FUNCTION_BLOCK FB_GCSpinAxisJogServices EXTENDS FB_PackMLBase IMPLEMENTS I_ModuleServiceProperty
VAR_INPUT
	Ctrl : REFERENCE TO ST_GCSpinAxisJogCtrl;
	Status : REFERENCE TO ST_GCSpinAxisJogStatus;
	Axis_BaseUnit : REFERENCE TO FB_AxisControl;
END_VAR

VAR_OUTPUT
END_VAR

VAR
	_StartOneShot	: R_TRIG;
	_ResetOneShot	: R_TRIG;
	_StopOneShot	: R_TRIG;
	_AbortOneShot	: R_TRIG;
	
	_ModuleMode		: T_PackMLMode;
END_VAR

// Update service state
Status.State := stOut.eStateCurrent;

A00_TrigCommand();

SUPER^();

ACTION A00_TrigCommand:
_StartOneShot(CLK:= Ctrl.Start);
IF _StartOneShot.Q THEN
	RequestCommand(E_PackMLCommand.Start);
END_IF

_ResetOneShot(CLK:= Ctrl.Reset);
IF _ResetOneShot.Q THEN
	RequestCommand(E_PackMLCommand.Reset);
END_IF

_StopOneShot(CLK:= Ctrl.Stop);
IF _StopOneShot.Q THEN
	RequestCommand(E_PackMLCommand.Stop);
END_IF

_AbortOneShot(CLK:= Ctrl.Abort);
IF _AbortOneShot.Q THEN
	RequestCommand(E_PackMLCommand.Abort);
END_IF
END_ACTION

METHOD PROTECTED H_OnAborted
VAR_INPUT
	bFirstScan	: BOOL;
END_VAR
// Default action hook intentionally empty. Override in derived FBs when needed.
Status.Busy := FALSE;
Status.Done := FALSE;
Status.Aborted := TRUE;

RequestCommand(E_PackMLCommand.Clear);
END_METHOD

METHOD PROTECTED H_OnAborting : E_PackMLHookResult
VAR_INPUT
	bFirstScan	: BOOL;
END_VAR
Axis_BaseUnit.M_Jog(
	JogForward:= FALSE, 
	JogBackwards:= FALSE, 
	Mode:= Ctrl.Param.Mode,
	Position:= Ctrl.Param.Position,
	Velocity:= Ctrl.Param.Velocity,
	Acceleration:= Ctrl.Param.Acceleration,
	Deceleration:= Ctrl.Param.Deceleration);

H_OnAborting := E_PackMLHookResult.Done;
END_METHOD

METHOD PROTECTED H_OnClearing : E_PackMLHookResult
VAR_INPUT
	bFirstScan	: BOOL;
END_VAR

VAR
	bServoOn : BOOL;
	bError : BOOL;
	nErrorId : UDINT;
END_VAR
H_OnClearing := E_PackMLHookResult.Done;
END_METHOD

METHOD PROTECTED H_OnComplete
VAR_INPUT
	bFirstScan	: BOOL;
END_VAR
Status.Busy := FALSE;
Status.Done := TRUE;
Status.Error := FALSE;
Status.Aborted := FALSE;
Status.ErrorId := E_GCSpinAxisJogErrorCode.None;

IF NOT Ctrl.Start THEN
	RequestCommand(E_PackMLCommand.Reset);
END_IF
END_METHOD

METHOD PROTECTED H_OnCompleting : E_PackMLHookResult
VAR_INPUT
	bFirstScan	: BOOL;
END_VAR
Status.Busy := FALSE;
Status.Done := TRUE;
Status.Error := FALSE;
Status.Aborted := FALSE;
Status.ErrorId := E_GCSpinAxisJogErrorCode.None;

Axis_BaseUnit.M_Jog(
	JogForward:= FALSE, 
	JogBackwards:= FALSE, 
	Mode:= Ctrl.Param.Mode,
	Position:= Ctrl.Param.Position,
	Velocity:= Ctrl.Param.Velocity,
	Acceleration:= Ctrl.Param.Acceleration,
	Deceleration:= Ctrl.Param.Deceleration);

H_OnCompleting := E_PackMLHookResult.Done;
END_METHOD

METHOD PROTECTED H_OnExecute : E_PackMLHookResult
VAR_INPUT
	bFirstScan	: BOOL;
END_VAR

VAR
	bDone : BOOL;
	bError : BOOL;
END_VAR
H_OnExecute := E_PackMLHookResult.Busy;

Status.Busy := TRUE;
Status.Done := FALSE;
Status.Error := FALSE;
Status.Aborted := FALSE;
Status.ErrorId := E_GCSpinAxisJogErrorCode.None;

Axis_BaseUnit.M_Jog(
	JogForward:= Ctrl.Param.JogForward,
	JogBackwards:= Ctrl.Param.JogBackwards,
	Mode:= Ctrl.Param.Mode,
	Position:= Ctrl.Param.Position,
	Velocity:= Ctrl.Param.Velocity,
	Acceleration:= Ctrl.Param.Acceleration,
	Deceleration:= Ctrl.Param.Deceleration,
	Done=> bDone, Error=> bError);


IF Ctrl.Param.Mode = E_JogMode.MC_JOGMODE_INCHING THEN
	IF bDone THEN
		Status.Busy := FALSE;
		Status.Done := TRUE;
		H_OnExecute := E_PackMLHookResult.Done;
		RETURN;
	END_IF
END_IF

IF bError THEN
		Status.Error := TRUE;
		Status.ErrorId := E_GCSpinAxisJogErrorCode.Jog_Error_During_Execute;
		
		RequestCommand(E_PackMLCommand.Stop);
END_IF
END_METHOD

METHOD PROTECTED H_OnHeld
VAR_INPUT
	bFirstScan	: BOOL;
END_VAR
// Default action hook intentionally empty. Override in derived FBs when needed.
END_METHOD

METHOD PROTECTED H_OnHolding : E_PackMLHookResult
VAR_INPUT
	bFirstScan	: BOOL;
END_VAR
// Default transient hooks complete immediately; override when work is required.
H_OnHolding := E_PackMLHookResult.Done;
END_METHOD

METHOD PROTECTED H_OnIdle
VAR_INPUT
	bFirstScan	: BOOL;
END_VAR
// Default action hook intentionally empty. Override in derived FBs when needed.
Status.Busy := FALSE;
Status.Done := FALSE;
Status.Error := FALSE;
Status.Aborted := FALSE;
Status.ErrorId := E_GCSpinAxisJogErrorCode.None;
END_METHOD

METHOD PROTECTED H_OnResetting : E_PackMLHookResult
VAR_INPUT
	bFirstScan	: BOOL;
END_VAR
Status.Busy := FALSE;
Status.Done := FALSE;
Status.Error := FALSE;
Status.Aborted := FALSE;
Status.ErrorId := E_GCSpinAxisJogErrorCode.None;

H_OnResetting := E_PackMLHookResult.Done;
END_METHOD

METHOD PROTECTED H_OnStarting : E_PackMLHookResult
VAR_INPUT
	bFirstScan	: BOOL;
END_VAR
H_OnStarting := E_PackMLHookResult.Busy;

Status.Busy := TRUE;
Status.Done := FALSE;
Status.Error := FALSE;
Status.Aborted := FALSE;
Status.ErrorId := E_GCSpinAxisJogErrorCode.None;

// Check is servo on
IF Axis_BaseUnit.AxisStatus.Disabled THEN
	
	// Throw up error
	Status.Error:= TRUE;
	Status.ErrorId:= E_GCSpinAxisJogErrorCode.Axis_Not_Servo_On_During_Starting;
	
	// Request abort command
	RequestCommand(E_PackMLCommand.Abort);
	RETURN;
END_IF

// Check is axis not busy
IF Axis_BaseUnit.AxisStatus.HasJob THEN
	// Throw up error
	Status.Error:= TRUE;
	Status.ErrorId:= E_GCSpinAxisJogErrorCode.Axis_Is_Busy_During_Starting;
	
	// Request abort command
	RequestCommand(E_PackMLCommand.Stop);
	RETURN;
END_IF

// Check is param valid
IF (Ctrl.Param.JogBackwards AND Ctrl.Param.JogForward) OR
	(NOT Ctrl.Param.JogBackwards AND NOT Ctrl.Param.JogForward) OR
	Ctrl.Param.Velocity = 0 THEN
	// Throw up error
	Status.Error:= TRUE;
	Status.ErrorId:= E_GCSpinAxisJogErrorCode.Invalid_Param;
	
	// Request abort command
	RequestCommand(E_PackMLCommand.Stop);
	RETURN;
END_IF

H_OnStarting := E_PackMLHookResult.Done;
END_METHOD

METHOD PROTECTED H_OnStopped
VAR_INPUT
	bFirstScan	: BOOL;
END_VAR
// Default action hook intentionally empty. Override in derived FBs when needed.
Status.Busy := FALSE;
Status.Done := FALSE;
Status.Aborted := TRUE;
END_METHOD

METHOD PROTECTED H_OnStopping : E_PackMLHookResult
VAR_INPUT
	bFirstScan	: BOOL;
END_VAR
Axis_BaseUnit.M_Jog(
	JogForward:= FALSE, 
	JogBackwards:= FALSE, 
	Mode:= Ctrl.Param.Mode,
	Position:= Ctrl.Param.Position,
	Velocity:= Ctrl.Param.Velocity,
	Acceleration:= Ctrl.Param.Acceleration,
	Deceleration:= Ctrl.Param.Deceleration);

H_OnStopping := E_PackMLHookResult.Done;
END_METHOD

METHOD PROTECTED H_OnSuspended
VAR_INPUT
	bFirstScan	: BOOL;
END_VAR
// Default action hook intentionally empty. Override in derived FBs when needed.
END_METHOD

METHOD PROTECTED H_OnSuspending : E_PackMLHookResult
VAR_INPUT
	bFirstScan	: BOOL;
END_VAR
// Default transient hooks complete immediately; override when work is required.
H_OnSuspending := E_PackMLHookResult.Done;
END_METHOD

METHOD PROTECTED H_OnUndefined : E_PackMLHookResult
VAR_INPUT
	bFirstScan	: BOOL;
END_VAR
// The base FB leaves Undefined immediately unless a derived FB delays startup.
H_OnUndefined := E_PackMLHookResult.Done;
END_METHOD

METHOD PROTECTED H_OnUnholding : E_PackMLHookResult
VAR_INPUT
	bFirstScan	: BOOL;
END_VAR
// Default transient hooks complete immediately; override when work is required.
H_OnUnholding := E_PackMLHookResult.Done;
END_METHOD

METHOD PROTECTED H_OnUnsuspending : E_PackMLHookResult
VAR_INPUT
	bFirstScan	: BOOL;
END_VAR
// Default transient hooks complete immediately; override when work is required.
H_OnUnsuspending := E_PackMLHookResult.Done;
END_METHOD

PROPERTY ModuleMode : T_PackMLMode
GET
ModuleMode := _ModuleMode;
END_GET
SET
_ModuleMode := ModuleMode;
END_SET
END_PROPERTY

END_FUNCTION_BLOCK

(* stored: Version 1.1.0.1, ProductVersion 3.1.4026.18
   POU FB_GCSpinAxisJogServices: Id {a61ac5cd-09b6-4f2d-bc54-d014db7401a2}, SpecialFunc None
   Folder StateAction: Id {30486db3-fa54-4a70-b426-5f8ba9d0504f}
   Action A00_TrigCommand: Id {d9012b4d-3f7d-455a-a3d6-1f5152c45f28}
   Method H_OnAborted: Id {b48428e2-059a-4878-a27b-576d41f2ba26}
   Method H_OnAborting: Id {df4c7f2d-8a88-4d35-a321-0716e918b536}
   Method H_OnClearing: Id {9a60118e-19f9-4bca-893b-e890bf0b19c9}
   Method H_OnComplete: Id {fd680a59-d09e-4091-ac1f-b02ebd6a48e6}
   Method H_OnCompleting: Id {61491643-adf6-4106-831a-f4dfe9e14738}
   Method H_OnExecute: Id {2dba6e2e-7918-46c6-a0b6-50da9e5cf338}
   Method H_OnHeld: Id {fc1df435-3bb5-4a7c-8ab6-c741096bcbf0}
   Method H_OnHolding: Id {ece160eb-a5c7-4980-a6c1-7b10ad25762b}
   Method H_OnIdle: Id {801e1204-bf1d-4d12-b7fd-e2791384226a}
   Method H_OnResetting: Id {cd0cb289-d0f8-442c-af15-52d2005bf619}
   Method H_OnStarting: Id {bcd7c333-82d2-481d-9c52-d49b2030a18e}
   Method H_OnStopped: Id {7643e72d-21d0-42a9-a466-1828d294ec10}
   Method H_OnStopping: Id {7e40e9e4-ecf0-49b7-86b3-13897394333e}
   Method H_OnSuspended: Id {e85e43db-649a-4658-a8a4-46ee44393ec1}
   Method H_OnSuspending: Id {e203e9d4-d997-4a54-8a42-be70e0403d06}
   Method H_OnUndefined: Id {f7603c5c-6fc0-49e6-83fe-7aacac7ddd39}
   Method H_OnUnholding: Id {273aa969-3e22-4ea9-8cb4-3dea54c7fc6d}
   Method H_OnUnsuspending: Id {901ae4a7-eddd-4729-903d-3db2ee99da23}
   Property ModuleMode: Id {909f5537-5629-4c46-9ccb-61a85ea831a5}
   Get Get: Id {e6b1fa22-a987-4664-8101-e14dca9a3d5a}
   Set Set: Id {4cdc4139-6e05-406a-b203-d0a353b0e373} *)
